PROGRAM PRG_02_Xdrive
VAR
	TOF_horn: TOF;
	bRipCut: BOOL;
	signal_light_blink_fwd: FB_Blinker;
	signal_light_blink_rev: FB_Blinker;
	signal_light_blink1: FB_Blinker;
	signal_light_blink2: FB_Blinker;
	R_TRIG_2: R_TRIG;
	R_TRIG_3: R_TRIG;
	bRemoteDRV :BOOL;
	bRemoteREV :BOOL;
	TOF_0: TOF;
	TOF_1: TOF;
	F_TRIG_0: F_TRIG;
	F_TRIG_1: F_TRIG;
END_VAR
VAR // added by the converter: edge detectors and wires of the graphical bodies
    _w1, _w2 : BOOL;
END_VAR

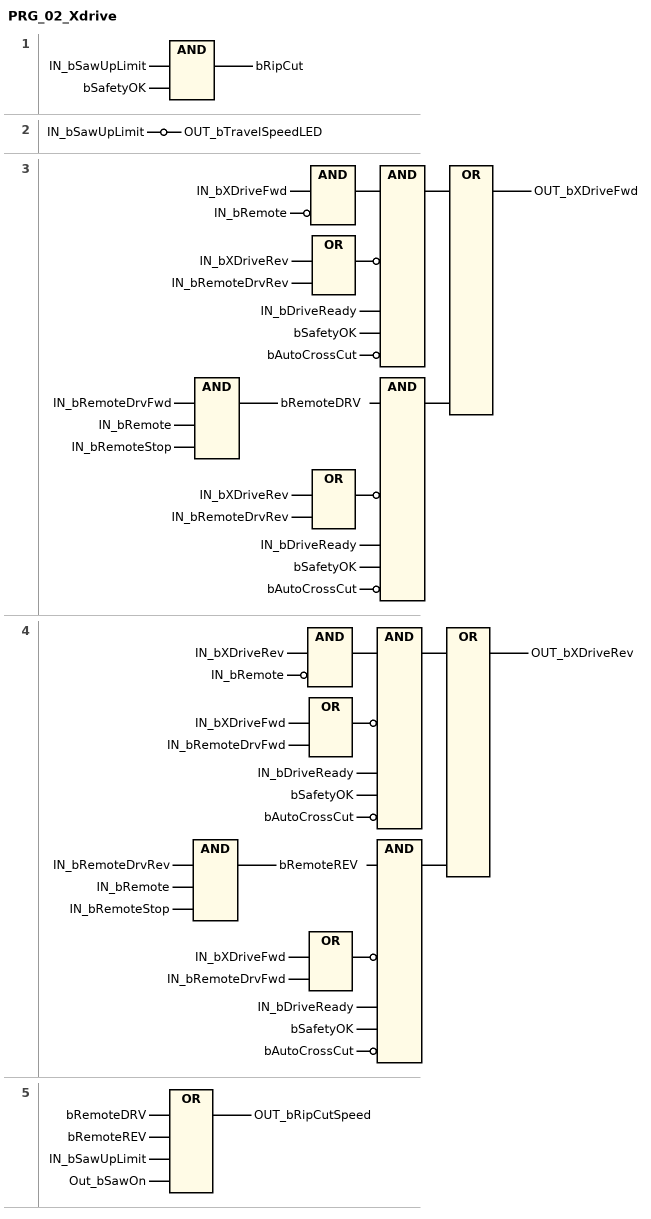
// NETWORK 1
bRipCut := IN_bSawUpLimit AND bSafetyOK;

// NETWORK 2
OUT_bTravelSpeedLED := NOT IN_bSawUpLimit;

// NETWORK 3
_w1 := IN_bRemoteDrvFwd AND IN_bRemote AND IN_bRemoteStop;
bRemoteDRV := _w1;
OUT_bXDriveFwd := (IN_bXDriveFwd AND NOT IN_bRemote) AND NOT (IN_bXDriveRev OR IN_bRemoteDrvRev) AND IN_bDriveReady AND bSafetyOK AND NOT bAutoCrossCut OR _w1 AND NOT (IN_bXDriveRev OR IN_bRemoteDrvRev) AND IN_bDriveReady AND bSafetyOK AND NOT bAutoCrossCut;

// NETWORK 4
_w2 := IN_bRemoteDrvRev AND IN_bRemote AND IN_bRemoteStop;
bRemoteREV := _w2;
OUT_bXDriveRev := (IN_bXDriveRev AND NOT IN_bRemote) AND NOT (IN_bXDriveFwd OR IN_bRemoteDrvFwd) AND IN_bDriveReady AND bSafetyOK AND NOT bAutoCrossCut OR _w2 AND NOT (IN_bXDriveFwd OR IN_bRemoteDrvFwd) AND IN_bDriveReady AND bSafetyOK AND NOT bAutoCrossCut;

// NETWORK 5
OUT_bRipCutSpeed := bRemoteDRV OR bRemoteREV OR IN_bSawUpLimit OR Out_bSawOn;

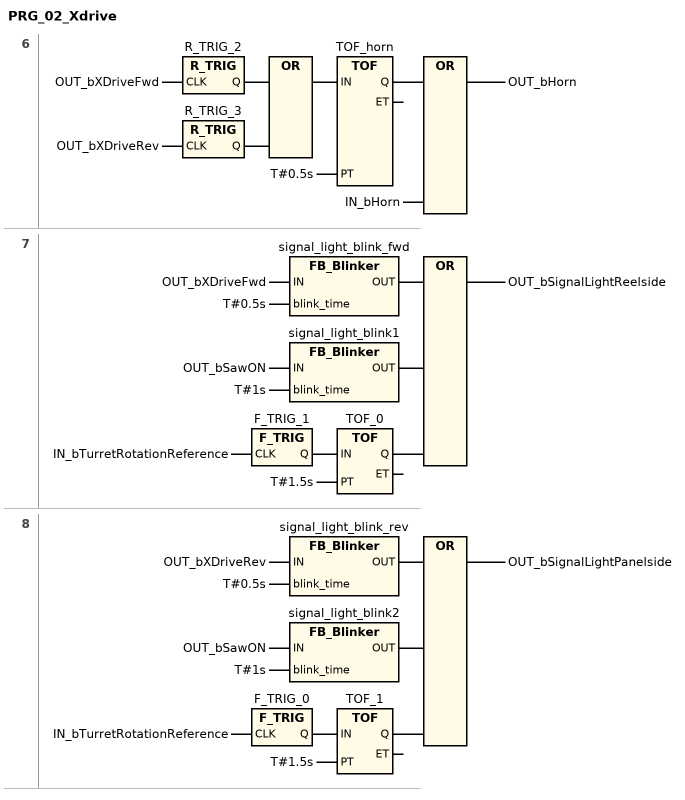
// NETWORK 6
R_TRIG_2(CLK := OUT_bXDriveFwd); // R_TRIG
R_TRIG_3(CLK := OUT_bXDriveRev); // R_TRIG
TOF_horn(IN := R_TRIG_2.Q OR R_TRIG_3.Q, PT := T#0.5s); // TOF
OUT_bHorn := TOF_horn.Q OR IN_bHorn;

// NETWORK 7
signal_light_blink_fwd(IN := OUT_bXDriveFwd, blink_time := T#0.5s); // FB_Blinker
signal_light_blink1(IN := OUT_bSawON, blink_time := T#1s); // FB_Blinker
F_TRIG_1(CLK := IN_bTurretRotationReference); // F_TRIG
TOF_0(IN := F_TRIG_1.Q, PT := T#1.5s); // TOF
OUT_bSignalLightReelside := signal_light_blink_fwd.OUT OR signal_light_blink1.OUT OR TOF_0.Q;

// NETWORK 8
signal_light_blink_rev(IN := OUT_bXDriveRev, blink_time := T#0.5s); // FB_Blinker
signal_light_blink2(IN := OUT_bSawON, blink_time := T#1s); // FB_Blinker
F_TRIG_0(CLK := IN_bTurretRotationReference); // F_TRIG
TOF_1(IN := F_TRIG_0.Q, PT := T#1.5s); // TOF
OUT_bSignalLightPanelside := signal_light_blink_rev.OUT OR signal_light_blink2.OUT OR TOF_1.Q;

END_PROGRAM

(* stored: Version 1.1.0.1, ProductVersion 3.1.4024.12
   POU PRG_02_Xdrive: Id {282c573b-0d0c-4cb8-981c-22f908547a63}, SpecialFunc None *)
